// TIA Portal V15.1 export
// export: Created 2024-05-17T05:38:36.8842157Z, ExportSetting WithDefaults, DisplayName Totally Integrated Automation Portal, DisplayVersion V15.1 Update 5, DisplayName TIA Portal Openness, DisplayVersion V15.1 Update 5, DisplayName SINAMICS Startdrive Advanced, DisplayVersion V15.1, DisplayName G130, G150, S120, S150, SINAMICS MV, S210, DisplayVersion V15.1, DisplayName G110M, G120, G120C, G120D, G120P, DisplayVersion V15.1, DisplayName STEP 7 Professional, DisplayVersion V15.1 Update 5, DisplayName STEP 7 Safety, DisplayVersion V15.1, DisplayName WinCC Professional, DisplayVersion V15.1 Update 5, DisplayName SIMATIC Visualization Architect, DisplayVersion V15.1
FUNCTION_BLOCK "LGBSEW-MoviFitFCPN"   // FB6620, FBD
TITLE = LSEW-MoviFitFCPN
{ S7_Optimized_Access := 'TRUE' }
AUTHOR : ENGIE
FAMILY : Actuator
VERSION : 0.1
// ============================================================================
// This module is the interface to a SEW drive MOVIFIT FC using telegram 003
// ============================================================================
// 
// SEW drive config:
// 
//  - 8.. Unit functions
//                   l - 87 Process data assignment
// 
//                                                                    _____________________
// 870 Setpoint description PO1              l Control word 2          v l
//                                                                    _____________________
// 871 Setpoint description PO2              l Setpoint speed [%]  v l
//                                                                    _____________________
// 872 Setpoint description PO3              l Ramp                          v l
//                                                                    _____________________
// 873 Actual value description PI1         l Status word 1            v l
//                                                                    _____________________
// 874 Actual value description PI2         l Output current          v l
//                                                                    _____________________
// 875 Actual value description PI3         l Status word 2            v l
//                                                                    _____________________
// 876 PO data enable                               l Yes                               v l 
//                                                                                      l
//                                                                                      v
//                                       This changes to no when a POx paramater is changed
//                                                 Dot not forget to put this back to yes !
// stored: AutoNumber false, IsIECCheckEnabled false, IsRetainMemResEnabled false, MemoryReserve 100, SetENOAutomatically False, UDAEnableTagReadback false
   VAR_INPUT
      I_ContolInhibit { ExternalAccessible := 'False'; ExternalVisible := 'False'; ExternalWritable := 'False'} : Bool;   // Inhibit motor (disable output stage, uncontolled stop)
      I_OFF1 { ExternalAccessible := 'False'; ExternalVisible := 'False'; ExternalWritable := 'False'} : Bool;   // start / stop motor
      I_OFF2 { ExternalAccessible := 'False'; ExternalVisible := 'False'; ExternalWritable := 'False'} : Bool := True;   // OFF2 rapid stop
      I_ResetFault { ExternalAccessible := 'False'; ExternalVisible := 'False'; ExternalWritable := 'False'} : Bool;   // Reset fault
      I_BrakeRelease { ExternalAccessible := 'False'; ExternalVisible := 'False'; ExternalWritable := 'False'} : Bool;   // Command brake release
      I_ParameterSet { ExternalAccessible := 'False'; ExternalVisible := 'False'; ExternalWritable := 'False'} : Bool;   // Select parameter set
      I_SetpointSpeed { ExternalAccessible := 'False'; ExternalVisible := 'False'; ExternalWritable := 'False'} : Real;   // Setpoint speed in -100-0-100%
      I_Ramp { ExternalAccessible := 'False'; ExternalVisible := 'False'; ExternalWritable := 'False'} : Time := T#1s;   // Ramp send in miliseconds (range : 100-10000ms, if 0 then default 1s will be used)
   END_VAR
   VAR_OUTPUT
      O_DriveReady { ExternalAccessible := 'False'; ExternalVisible := 'False'; ExternalWritable := 'False'} : Bool;   // Drive ready
      O_OutputStageEnabled { ExternalAccessible := 'False'; ExternalVisible := 'False'; ExternalWritable := 'False'} : Bool;   // Inverter output stage is enabled
      O_MaintenanceSwitch { ExternalAccessible := 'False'; ExternalVisible := 'False'; ExternalWritable := 'False'} : Bool;   // Maintenance switch activated (1=mains OFF)
      O_ParameterSet { ExternalAccessible := 'False'; ExternalVisible := 'False'; ExternalWritable := 'False'} : Bool;   // Active parameter set
      O_PODataEnabled { ExternalAccessible := 'False'; ExternalVisible := 'False'; ExternalWritable := 'False'} : Bool;   // Process data is enabled (1 = Drive can be controlled via fieldbus)
      O_Fault { ExternalAccessible := 'False'; ExternalVisible := 'False'; ExternalWritable := 'False'} : Bool;   // Fault present
      O_Brake { ExternalAccessible := 'False'; ExternalVisible := 'False'; ExternalWritable := 'False'} : Bool;   // Brake status
      O_ActorVoltageOverloadDO00 { ExternalAccessible := 'False'; ExternalVisible := 'False'; ExternalWritable := 'False'} : Bool;   // Short circuit / overload of the actuator voltage for digital output DO00
      O_ActorVoltageOverloadDO01 { ExternalAccessible := 'False'; ExternalVisible := 'False'; ExternalWritable := 'False'} : Bool;   // Short circuit / overload of the actuator voltage for digital output DO01
      O_ActorVoltageOverloadDO02 { ExternalAccessible := 'False'; ExternalVisible := 'False'; ExternalWritable := 'False'} : Bool;   // Short circuit / overload of the actuator voltage for digital output DO02
      O_ActorVoltageOverloadDO03 { ExternalAccessible := 'False'; ExternalVisible := 'False'; ExternalWritable := 'False'} : Bool;   // Short circuit / overload of the actuator voltage for digital output DO03
      O_SensorVoltageOverloadGroup1 { ExternalAccessible := 'False'; ExternalVisible := 'False'; ExternalWritable := 'False'} : Bool;   // Short circuit / overload of the sensor suuply group 1 (VO24-I)
      O_SensorVoltageOverloadGroup2 { ExternalAccessible := 'False'; ExternalVisible := 'False'; ExternalWritable := 'False'} : Bool;   // Short circuit / overload of the sensor suuply group 2 (VO24-I)
      O_SensorVoltageOverloadGroup3 { ExternalAccessible := 'False'; ExternalVisible := 'False'; ExternalWritable := 'False'} : Bool;   // Short circuit / overload of the sensor suuply group 3 (VO24-I)
      O_SensorVoltageOverloadGroup4 { ExternalAccessible := 'False'; ExternalVisible := 'False'; ExternalWritable := 'False'} : Bool;   // Short circuit / overload of the sensor suuply group 4 (VO24-I)
      "O_Undervoltage24V-S" { ExternalAccessible := 'False'; ExternalVisible := 'False'; ExternalWritable := 'False'} : Bool;   // Value falls below the power limit for the actuator voltage DO00-03
      "O_InverterVoltageNotApplied24V-P" { ExternalAccessible := 'False'; ExternalVisible := 'False'; ExternalWritable := 'False'} : Bool;   // Presence of 24V_P for integrated inverter (FC) or external MOVIMOT (1=24V_P not present)
      O_MOVIFITSystemFault { ExternalAccessible := 'False'; ExternalVisible := 'False'; ExternalWritable := 'False'} : Bool;   // MOVIFIT system fault
      H_StatusWord1 { ExternalAccessible := 'False'; ExternalVisible := 'False'; ExternalWritable := 'False'} : Word;   // Status word 1 from drive
      H_StatusWord2 { ExternalAccessible := 'False'; ExternalVisible := 'False'; ExternalWritable := 'False'} : Word;   // Status word 2 from drive
      H_StatusWord3 { ExternalAccessible := 'False'; ExternalVisible := 'False'; ExternalWritable := 'False'} : Word;   // Status word 3 from drive
      H_ControlWord { ExternalAccessible := 'False'; ExternalVisible := 'False'; ExternalWritable := 'False'} : Word;   // Control word to drive
      H_SetpointSpeed { ExternalAccessible := 'False'; ExternalVisible := 'False'; ExternalWritable := 'False'} : Word;   // Speed setpoint for drive
      H_SetpointSpeedProCent { ExternalAccessible := 'False'; ExternalVisible := 'False'; ExternalWritable := 'False'} : Real;   // Speed setpoint for drive % / Speed setpoint for drive
      H_SetpointRamp { ExternalAccessible := 'False'; ExternalVisible := 'False'; ExternalWritable := 'False'} : Int;   // Ramp setpoint for drive
      H_ActualCurrentA { ExternalAccessible := 'False'; ExternalVisible := 'False'; ExternalWritable := 'False'} : Real;   // Actual current Ampere
      H_ActualCurrentProCent { ExternalAccessible := 'False'; ExternalVisible := 'False'; ExternalWritable := 'False'} : Real;   // Actual current %
      H_ActualWarning { ExternalAccessible := 'False'; ExternalVisible := 'False'; ExternalWritable := 'False'} : Int;   // Actual Warning From Drive
      H_ActualFault { ExternalAccessible := 'False'; ExternalVisible := 'False'; ExternalWritable := 'False'} : Int;   // Actual Fault From Drive
   END_VAR
   VAR_IN_OUT
      C_HWSubInput { ExternalAccessible := 'False'; ExternalVisible := 'False'; ExternalWritable := 'False'} : HW_SUBMODULE;   // Inputs telegram 3 Hardware identifier
      C_HWSubInputStatus { ExternalAccessible := 'False'; ExternalVisible := 'False'; ExternalWritable := 'False'} : HW_SUBMODULE;   // Status telegram MOVIFIT Hardware identifier
      C_HWSubOutput { ExternalAccessible := 'False'; ExternalVisible := 'False'; ExternalWritable := 'False'} : HW_SUBMODULE;   // Outputs telegram 3 Hardware identifier
      C_DriveCurrent { ExternalAccessible := 'False'; ExternalVisible := 'False'; ExternalWritable := 'False'} : Real;   // Reference current of the drive
      C_MotorCurrent { ExternalAccessible := 'False'; ExternalVisible := 'False'; ExternalWritable := 'False'} : Real;   // Reference current of the motor
   END_VAR
   VAR
      InputTelegram { ExternalAccessible := 'False'; ExternalVisible := 'False'; ExternalWritable := 'False'} : Struct   // Inputs telegram 3
         PI1 { ExternalAccessible := 'False'; ExternalVisible := 'False'; ExternalWritable := 'False'} : Struct   // Status word 1
            Status { ExternalAccessible := 'False'; ExternalVisible := 'False'; ExternalWritable := 'False'} : Byte;   // Status / error code
            OutputStageEnabled { ExternalAccessible := 'False'; ExternalVisible := 'False'; ExternalWritable := 'False'} : Bool;   // Inverter output stage is enabled
            InverterReady { ExternalAccessible := 'False'; ExternalVisible := 'False'; ExternalWritable := 'False'} : Bool;   // Inverter power section is ready for operation
            PODataEnabled { ExternalAccessible := 'False'; ExternalVisible := 'False'; ExternalWritable := 'False'} : Bool;   // Process data is enabled (1 = Drive can be controlled via fieldbus)
            Spare1 { ExternalAccessible := 'False'; ExternalVisible := 'False'; ExternalWritable := 'False'} : Bool;   // Reserved / not used
            CurrentParSet { ExternalAccessible := 'False'; ExternalVisible := 'False'; ExternalWritable := 'False'} : Bool;   // Current parameter set
            FaultWarning { ExternalAccessible := 'False'; ExternalVisible := 'False'; ExternalWritable := 'False'} : Bool;   // Fault/warning present
            Spare2 { ExternalAccessible := 'False'; ExternalVisible := 'False'; ExternalWritable := 'False'} : Bool;   // Reserved / not used
            Spare3 { ExternalAccessible := 'False'; ExternalVisible := 'False'; ExternalWritable := 'False'} : Bool;   // Reserved / not used
         END_STRUCT;
         Current { ExternalAccessible := 'False'; ExternalVisible := 'False'; ExternalWritable := 'False'} : Int;   // Current
         PI3 { ExternalAccessible := 'False'; ExternalVisible := 'False'; ExternalWritable := 'False'} : Struct   // Status word 2
            brake { ExternalAccessible := 'False'; ExternalVisible := 'False'; ExternalWritable := 'False'} : Bool;   // Brake released
            Spare4 { ExternalAccessible := 'False'; ExternalVisible := 'False'; ExternalWritable := 'False'} : Bool;   // Reserved / not used
            Spare5 { ExternalAccessible := 'False'; ExternalVisible := 'False'; ExternalWritable := 'False'} : Bool;   // Reserved / not used
            Spare6 { ExternalAccessible := 'False'; ExternalVisible := 'False'; ExternalWritable := 'False'} : Bool;   // Reserved / not used
            Spare7 { ExternalAccessible := 'False'; ExternalVisible := 'False'; ExternalWritable := 'False'} : Bool;   // Reserved / not used
            Spare8 { ExternalAccessible := 'False'; ExternalVisible := 'False'; ExternalWritable := 'False'} : Bool;   // Reserved / not used
            Spare9 { ExternalAccessible := 'False'; ExternalVisible := 'False'; ExternalWritable := 'False'} : Bool;   // Reserved / not used
            Spare10 { ExternalAccessible := 'False'; ExternalVisible := 'False'; ExternalWritable := 'False'} : Bool;   // Reserved / not used
            OutputStageEnabled { ExternalAccessible := 'False'; ExternalVisible := 'False'; ExternalWritable := 'False'} : Bool;   // Inverter output stage is enabled
            InverterReady { ExternalAccessible := 'False'; ExternalVisible := 'False'; ExternalWritable := 'False'} : Bool;   // Inverter power section is ready for operation
            PODataEnabled { ExternalAccessible := 'False'; ExternalVisible := 'False'; ExternalWritable := 'False'} : Bool;   // Process data is enabled (1 = Drive can be controlled via fieldbus)
            Spare11 { ExternalAccessible := 'False'; ExternalVisible := 'False'; ExternalWritable := 'False'} : Bool;   // Reserved / not used
            CurrentParSet { ExternalAccessible := 'False'; ExternalVisible := 'False'; ExternalWritable := 'False'} : Bool;   // Current parameter set
            FaultWarning { ExternalAccessible := 'False'; ExternalVisible := 'False'; ExternalWritable := 'False'} : Bool;   // Fault/warning present
            Spare12 { ExternalAccessible := 'False'; ExternalVisible := 'False'; ExternalWritable := 'False'} : Bool;   // Reserved / not used
            Spare13 { ExternalAccessible := 'False'; ExternalVisible := 'False'; ExternalWritable := 'False'} : Bool;   // Reserved / not used
         END_STRUCT;
      END_STRUCT;
      InputStatusTelegram { ExternalAccessible := 'False'; ExternalVisible := 'False'; ExternalWritable := 'False'} : Struct   // Status telegram MOVIFIT
         ActorVoltageOverloadDO00 { ExternalAccessible := 'False'; ExternalVisible := 'False'; ExternalWritable := 'False'} : Bool;   // Short circuit / overload of the actuator voltage for digital output DO00
         ActorVoltageOverloadDO01 { ExternalAccessible := 'False'; ExternalVisible := 'False'; ExternalWritable := 'False'} : Bool;   // Short circuit / overload of the actuator voltage for digital output DO01
         ActorVoltageOverloadDO02 { ExternalAccessible := 'False'; ExternalVisible := 'False'; ExternalWritable := 'False'} : Bool;   // Short circuit / overload of the actuator voltage for digital output DO02
         ActorVoltageOverloadDO03 { ExternalAccessible := 'False'; ExternalVisible := 'False'; ExternalWritable := 'False'} : Bool;   // Short circuit / overload of the actuator voltage for digital output DO03
         SensorVoltageOverloadGroup1 { ExternalAccessible := 'False'; ExternalVisible := 'False'; ExternalWritable := 'False'} : Bool;   // Short circuit / overload of the sensor suuply group 1 (VO24-I)
         SensorVoltageOverloadGroup2 { ExternalAccessible := 'False'; ExternalVisible := 'False'; ExternalWritable := 'False'} : Bool;   // Short circuit / overload of the sensor suuply group 2 (VO24-I)
         SensorVoltageOverloadGroup3 { ExternalAccessible := 'False'; ExternalVisible := 'False'; ExternalWritable := 'False'} : Bool;   // Short circuit / overload of the sensor suuply group 3 (VO24-I)
         SensorVoltageOverloadGroup4 { ExternalAccessible := 'False'; ExternalVisible := 'False'; ExternalWritable := 'False'} : Bool;   // Short circuit / overload of the sensor suuply group 4 (VO24-I)
         MaintenanceSwitch { ExternalAccessible := 'False'; ExternalVisible := 'False'; ExternalWritable := 'False'} : Bool;   // Maintenance switch activated (1=mains OFF)
         "Undervoltage24V-S" { ExternalAccessible := 'False'; ExternalVisible := 'False'; ExternalWritable := 'False'} : Bool;   // Value falls below the power limit for the actuator voltage DO00-03
         "InverterVoltageNotApplied24V-P" { ExternalAccessible := 'False'; ExternalVisible := 'False'; ExternalWritable := 'False'} : Bool;   // Presence of 24V_P for integrated inverter (FC) or external MOVIMOT (1=24V_P not present)
         Spare1 { ExternalAccessible := 'False'; ExternalVisible := 'False'; ExternalWritable := 'False'} : Bool;   // Reserved / not used
         Spare2 { ExternalAccessible := 'False'; ExternalVisible := 'False'; ExternalWritable := 'False'} : Bool;   // Reserved / not used
         Spare3 { ExternalAccessible := 'False'; ExternalVisible := 'False'; ExternalWritable := 'False'} : Bool;   // Reserved / not used
         Spare4 { ExternalAccessible := 'False'; ExternalVisible := 'False'; ExternalWritable := 'False'} : Bool;   // Reserved / not used
         MOVIFITSystemFault { ExternalAccessible := 'False'; ExternalVisible := 'False'; ExternalWritable := 'False'} : Bool;   // MOVIFIT system fault
      END_STRUCT;
      OutputTelegram { ExternalAccessible := 'False'; ExternalVisible := 'False'; ExternalWritable := 'False'} : Struct   // Outputs telegram 3
         PO1 { ExternalAccessible := 'False'; ExternalVisible := 'False'; ExternalWritable := 'False'} : Struct
            BrakeRelease { ExternalAccessible := 'False'; ExternalVisible := 'False'; ExternalWritable := 'False'} : Bool;   // Release brake
            CTW_Bit9 { ExternalAccessible := 'False'; ExternalVisible := 'False'; ExternalWritable := 'False'} : Bool;   // Reserved / not used
            CTW_Bit10 { ExternalAccessible := 'False'; ExternalVisible := 'False'; ExternalWritable := 'False'} : Bool;   // Reserved / not used
            CTW_Bit11 { ExternalAccessible := 'False'; ExternalVisible := 'False'; ExternalWritable := 'False'} : Bool;   // Reserved / not used
            CTW_Bit12 { ExternalAccessible := 'False'; ExternalVisible := 'False'; ExternalWritable := 'False'} : Bool;   // Reserved / not used
            CTW_Bit13 { ExternalAccessible := 'False'; ExternalVisible := 'False'; ExternalWritable := 'False'} : Bool;   // Reserved / not used
            CTW_Bit14 { ExternalAccessible := 'False'; ExternalVisible := 'False'; ExternalWritable := 'False'} : Bool;   // Reserved / not used
            CTW_Bit15 { ExternalAccessible := 'False'; ExternalVisible := 'False'; ExternalWritable := 'False'} : Bool;   // Reserved / not used
            ContrInhibit { ExternalAccessible := 'False'; ExternalVisible := 'False'; ExternalWritable := 'False'} : Bool;   // Interlock to drive
            RapidStop { ExternalAccessible := 'False'; ExternalVisible := 'False'; ExternalWritable := 'False'} : Bool;   // Rapid stop with stop ramp t13/t23, brake applied after stop
            Stop { ExternalAccessible := 'False'; ExternalVisible := 'False'; ExternalWritable := 'False'} : Bool;   // Stop to drive at normal ramp
            CTW_Bit3 { ExternalAccessible := 'False'; ExternalVisible := 'False'; ExternalWritable := 'False'} : Bool;   // Reserved / not used
            CTW_Bit4 { ExternalAccessible := 'False'; ExternalVisible := 'False'; ExternalWritable := 'False'} : Bool;   // Reserved / not used
            CTW_Bit5 { ExternalAccessible := 'False'; ExternalVisible := 'False'; ExternalWritable := 'False'} : Bool;   // Reserved / not used / Parameter set 1 or 2
            ResetFault { ExternalAccessible := 'False'; ExternalVisible := 'False'; ExternalWritable := 'False'} : Bool;   // Reset fault on drive
            CTW_Bit7 { ExternalAccessible := 'False'; ExternalVisible := 'False'; ExternalWritable := 'False'} : Bool;   // Reserved / not used
         END_STRUCT;
         SetpointSpeed { ExternalAccessible := 'False'; ExternalVisible := 'False'; ExternalWritable := 'False'} : Word;   // Speed setpoint for drive (-4000-0-4000hex)
         Ramp { ExternalAccessible := 'False'; ExternalVisible := 'False'; ExternalWritable := 'False'} : Int;   // Ramp setpoint for drive
      END_STRUCT;
   END_VAR
   VAR_TEMP
      TempReal : Real;   // Temp Real
   END_VAR
   VAR_TEMP   // added for the SCL form of the ladder/FBD networks
      _w1 : Bool;
   END_VAR
BEGIN

REGION Network 1: **** 1 - Inputs **** Read input telegram and store in struct
   // Copies the Input telegram to a local varibale struct
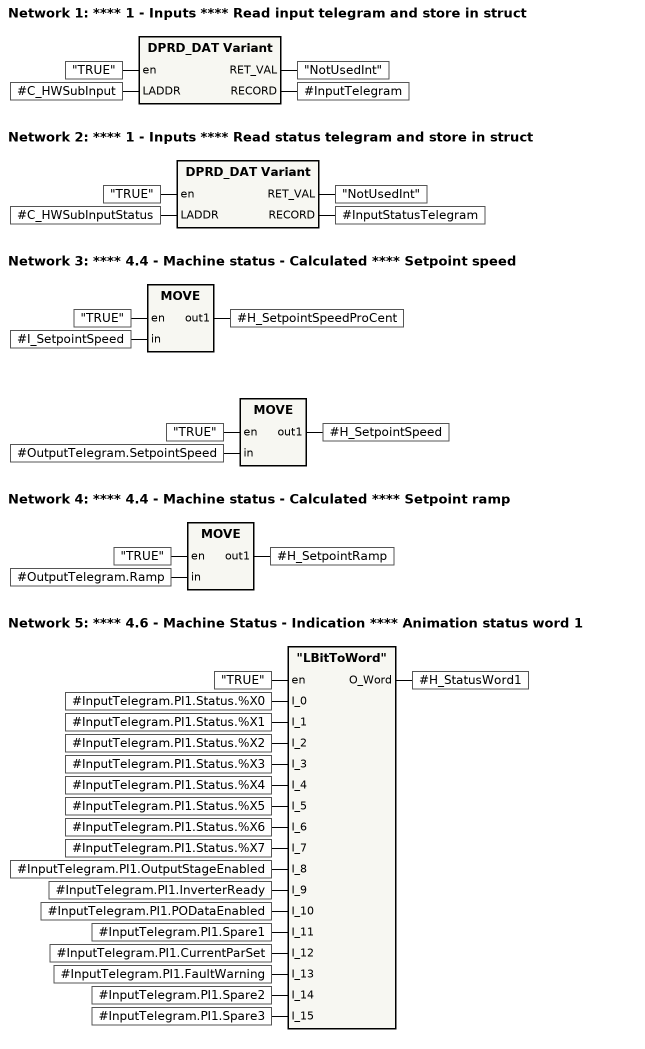
   IF "TRUE" THEN
       "NotUsedInt" := DPRD_DAT(LADDR := #C_HWSubInput, RECORD => #InputTelegram);   // Copy data with HW ID _________ /________ / l input telegram l SEW l l ===============>> PLC l Drive _l / -l__l
   END_IF;
END_REGION

REGION Network 2: **** 1 - Inputs **** Read status telegram and store in struct
   // Copies the status telegram to a local varibale struct
   IF "TRUE" THEN
       "NotUsedInt" := DPRD_DAT(LADDR := #C_HWSubInputStatus, RECORD => #InputStatusTelegram);   // Copy data with HW ID _________ /________ / l Status telegram l SEW l l ===============>> PLC l Drive _l / -l__l
   END_IF;
END_REGION

REGION Network 3: **** 4.4 - Machine status - Calculated **** Setpoint speed
   // Convert Data
   IF "TRUE" THEN
       #H_SetpointSpeedProCent := #I_SetpointSpeed;
       #H_SetpointSpeed := #OutputTelegram.SetpointSpeed;
   END_IF;
END_REGION

REGION Network 4: **** 4.4 - Machine status - Calculated **** Setpoint ramp
   // Convert Data
   IF "TRUE" THEN #H_SetpointRamp := #OutputTelegram.Ramp; END_IF;
END_REGION

REGION Network 5: **** 4.6 - Machine Status - Indication **** Animation status word 1
   // Animation
   IF "TRUE" THEN
       "LBitToWord"(I_0 := #InputTelegram.PI1.Status.%X0,
                    I_1 := #InputTelegram.PI1.Status.%X1,
                    I_2 := #InputTelegram.PI1.Status.%X2,
                    I_3 := #InputTelegram.PI1.Status.%X3,
                    I_4 := #InputTelegram.PI1.Status.%X4,
                    I_5 := #InputTelegram.PI1.Status.%X5,
                    I_6 := #InputTelegram.PI1.Status.%X6,
                    I_7 := #InputTelegram.PI1.Status.%X7,
                    I_8 := #InputTelegram.PI1.OutputStageEnabled,
                    I_9 := #InputTelegram.PI1.InverterReady,
                    I_10 := #InputTelegram.PI1.PODataEnabled,
                    I_11 := #InputTelegram.PI1.Spare1,
                    I_12 := #InputTelegram.PI1.CurrentParSet,
                    I_13 := #InputTelegram.PI1.FaultWarning,
                    I_14 := #InputTelegram.PI1.Spare2,
                    I_15 := #InputTelegram.PI1.Spare3,
                    O_Word => #H_StatusWord1);
   END_IF;
END_REGION

REGION Network 6: **** 4.6 - Machine Status - Indication **** Animation status word 2
   // Animation
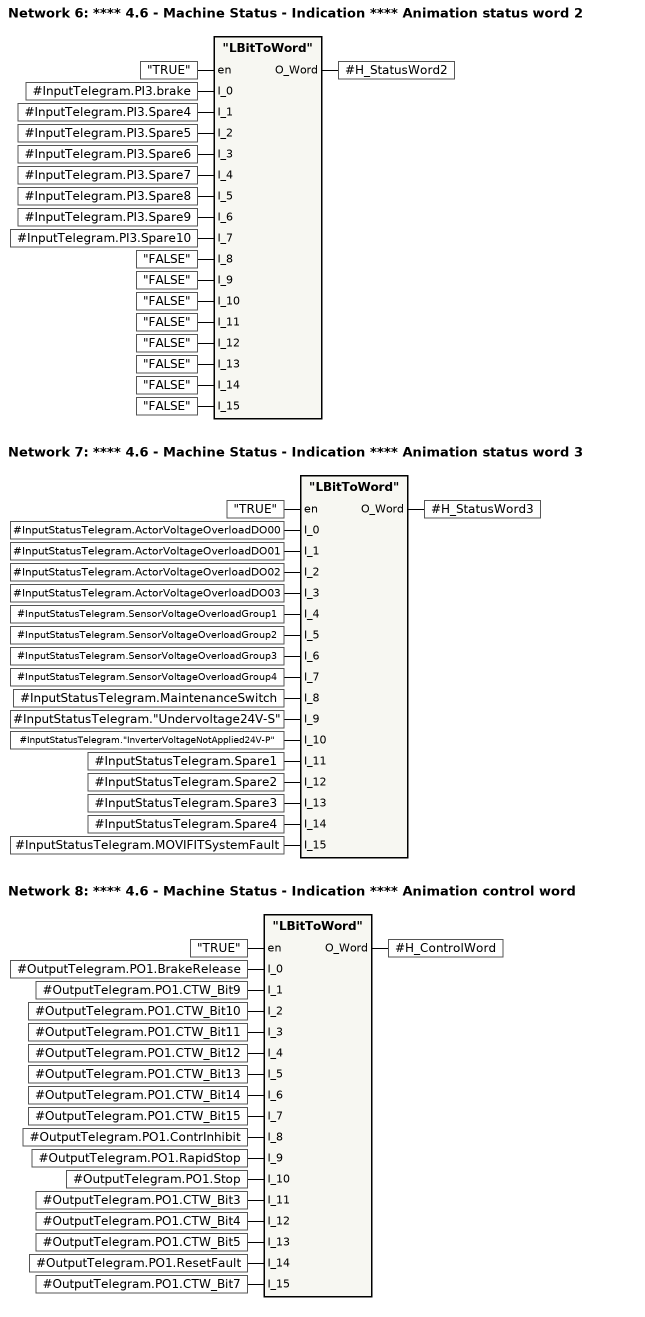
   IF "TRUE" THEN
       "LBitToWord"(I_0 := #InputTelegram.PI3.brake,
                    I_1 := #InputTelegram.PI3.Spare4,
                    I_2 := #InputTelegram.PI3.Spare5,
                    I_3 := #InputTelegram.PI3.Spare6,
                    I_4 := #InputTelegram.PI3.Spare7,
                    I_5 := #InputTelegram.PI3.Spare8,
                    I_6 := #InputTelegram.PI3.Spare9,
                    I_7 := #InputTelegram.PI3.Spare10,
                    I_8 := "FALSE",
                    I_9 := "FALSE",
                    I_10 := "FALSE",
                    I_11 := "FALSE",
                    I_12 := "FALSE",
                    I_13 := "FALSE",
                    I_14 := "FALSE",
                    I_15 := "FALSE",
                    O_Word => #H_StatusWord2);
   END_IF;
END_REGION

REGION Network 7: **** 4.6 - Machine Status - Indication **** Animation status word 3
   // Animation
   IF "TRUE" THEN
       "LBitToWord"(I_0 := #InputStatusTelegram.ActorVoltageOverloadDO00,
                    I_1 := #InputStatusTelegram.ActorVoltageOverloadDO01,
                    I_2 := #InputStatusTelegram.ActorVoltageOverloadDO02,
                    I_3 := #InputStatusTelegram.ActorVoltageOverloadDO03,
                    I_4 := #InputStatusTelegram.SensorVoltageOverloadGroup1,
                    I_5 := #InputStatusTelegram.SensorVoltageOverloadGroup2,
                    I_6 := #InputStatusTelegram.SensorVoltageOverloadGroup3,
                    I_7 := #InputStatusTelegram.SensorVoltageOverloadGroup4,
                    I_8 := #InputStatusTelegram.MaintenanceSwitch,
                    I_9 := #InputStatusTelegram."Undervoltage24V-S",
                    I_10 := #InputStatusTelegram."InverterVoltageNotApplied24V-P",
                    I_11 := #InputStatusTelegram.Spare1,
                    I_12 := #InputStatusTelegram.Spare2,
                    I_13 := #InputStatusTelegram.Spare3,
                    I_14 := #InputStatusTelegram.Spare4,
                    I_15 := #InputStatusTelegram.MOVIFITSystemFault,
                    O_Word => #H_StatusWord3);
   END_IF;
END_REGION

REGION Network 8: **** 4.6 - Machine Status - Indication **** Animation control word
   // Animation
   IF "TRUE" THEN
       "LBitToWord"(I_0 := #OutputTelegram.PO1.BrakeRelease,
                    I_1 := #OutputTelegram.PO1.CTW_Bit9,
                    I_2 := #OutputTelegram.PO1.CTW_Bit10,
                    I_3 := #OutputTelegram.PO1.CTW_Bit11,
                    I_4 := #OutputTelegram.PO1.CTW_Bit12,
                    I_5 := #OutputTelegram.PO1.CTW_Bit13,
                    I_6 := #OutputTelegram.PO1.CTW_Bit14,
                    I_7 := #OutputTelegram.PO1.CTW_Bit15,
                    I_8 := #OutputTelegram.PO1.ContrInhibit,
                    I_9 := #OutputTelegram.PO1.RapidStop,
                    I_10 := #OutputTelegram.PO1.Stop,
                    I_11 := #OutputTelegram.PO1.CTW_Bit3,
                    I_12 := #OutputTelegram.PO1.CTW_Bit4,
                    I_13 := #OutputTelegram.PO1.CTW_Bit5,
                    I_14 := #OutputTelegram.PO1.ResetFault,
                    I_15 := #OutputTelegram.PO1.CTW_Bit7,
                    O_Word => #H_ControlWord);
   END_IF;
END_REGION

REGION Network 9: **** 4.6 - Machine Status - Calculated **** Status / Warning / Fault code from drive
   // When the fault input is "True"   then the status code send over the byte is a fault code as decimal.
   // When the fault input is "False" then the status code send over the byte is a warning / status code as decimal.
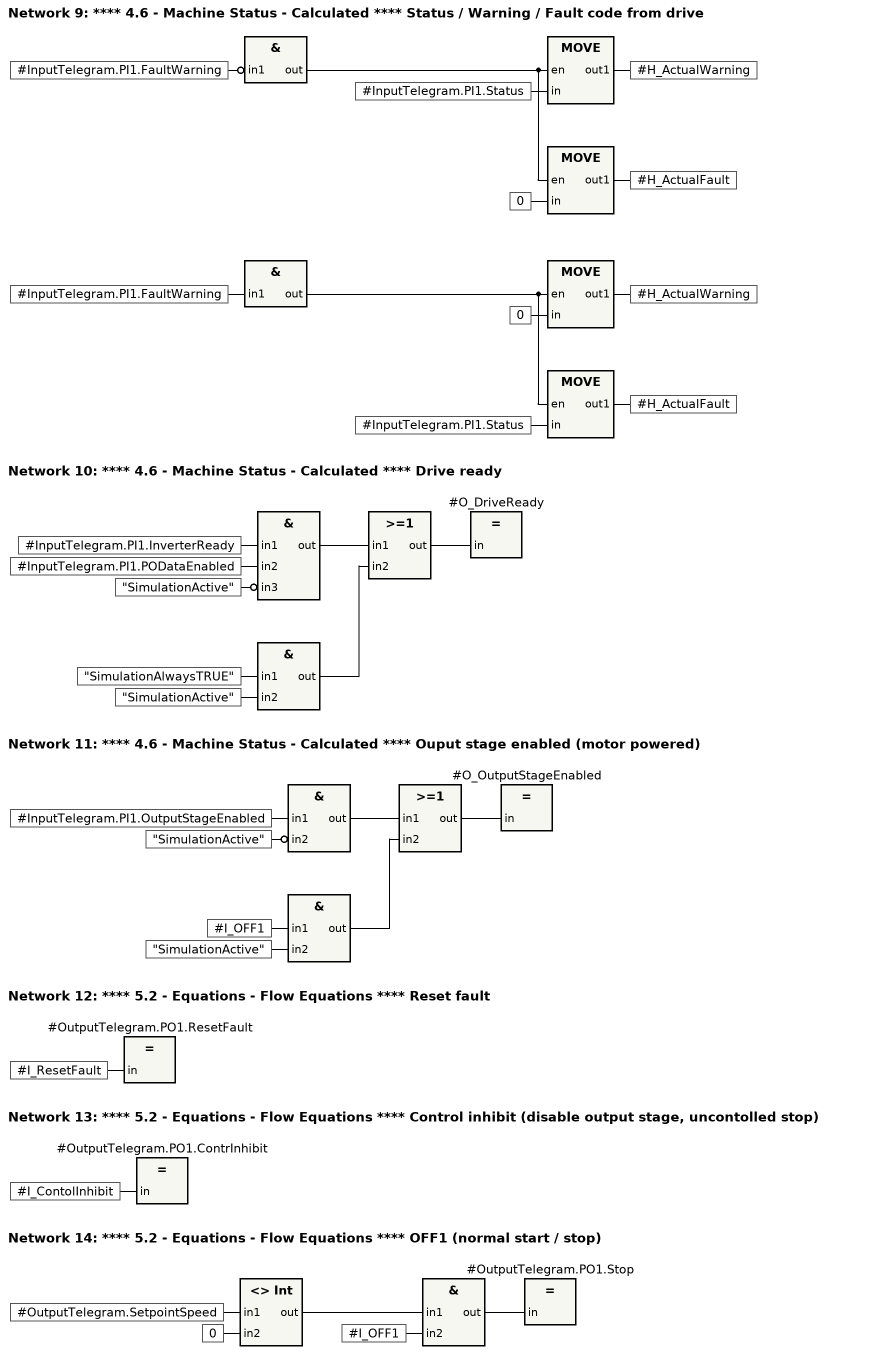
   IF NOT #InputTelegram.PI1.FaultWarning THEN
       #H_ActualWarning := #InputTelegram.PI1.Status;
       #H_ActualFault := 0;
   END_IF;
   IF #InputTelegram.PI1.FaultWarning THEN
       #H_ActualWarning := 0;
       #H_ActualFault := #InputTelegram.PI1.Status;
   END_IF;
END_REGION

REGION Network 10: **** 4.6 - Machine Status - Calculated **** Drive ready
   // Drive ready state and process data from PLC is active (Drive is listening to PLC)
   #O_DriveReady := (#InputTelegram.PI1.InverterReady AND #InputTelegram.PI1.PODataEnabled AND NOT "SimulationActive") OR ("SimulationAlwaysTRUE" AND "SimulationActive");
END_REGION

REGION Network 11: **** 4.6 - Machine Status - Calculated **** Ouput stage enabled (motor powered)
   // Ouput stage enabled (motor powered)
   #O_OutputStageEnabled := (#InputTelegram.PI1.OutputStageEnabled AND NOT "SimulationActive") OR (#I_OFF1 AND "SimulationActive");
END_REGION

REGION Network 12: **** 5.2 - Equations - Flow Equations **** Reset fault
   #OutputTelegram.PO1.ResetFault := #I_ResetFault;
END_REGION

REGION Network 13: **** 5.2 - Equations - Flow Equations **** Control inhibit (disable output stage, uncontolled stop)
   #OutputTelegram.PO1.ContrInhibit := #I_ContolInhibit;
END_REGION

REGION Network 14: **** 5.2 - Equations - Flow Equations **** OFF1 (normal start / stop)
   #OutputTelegram.PO1.Stop := (#OutputTelegram.SetpointSpeed <> 0) AND #I_OFF1;
END_REGION

REGION Network 15: **** 5.2 - Equations - Flow Equations **** OFF2 (rapid stop)
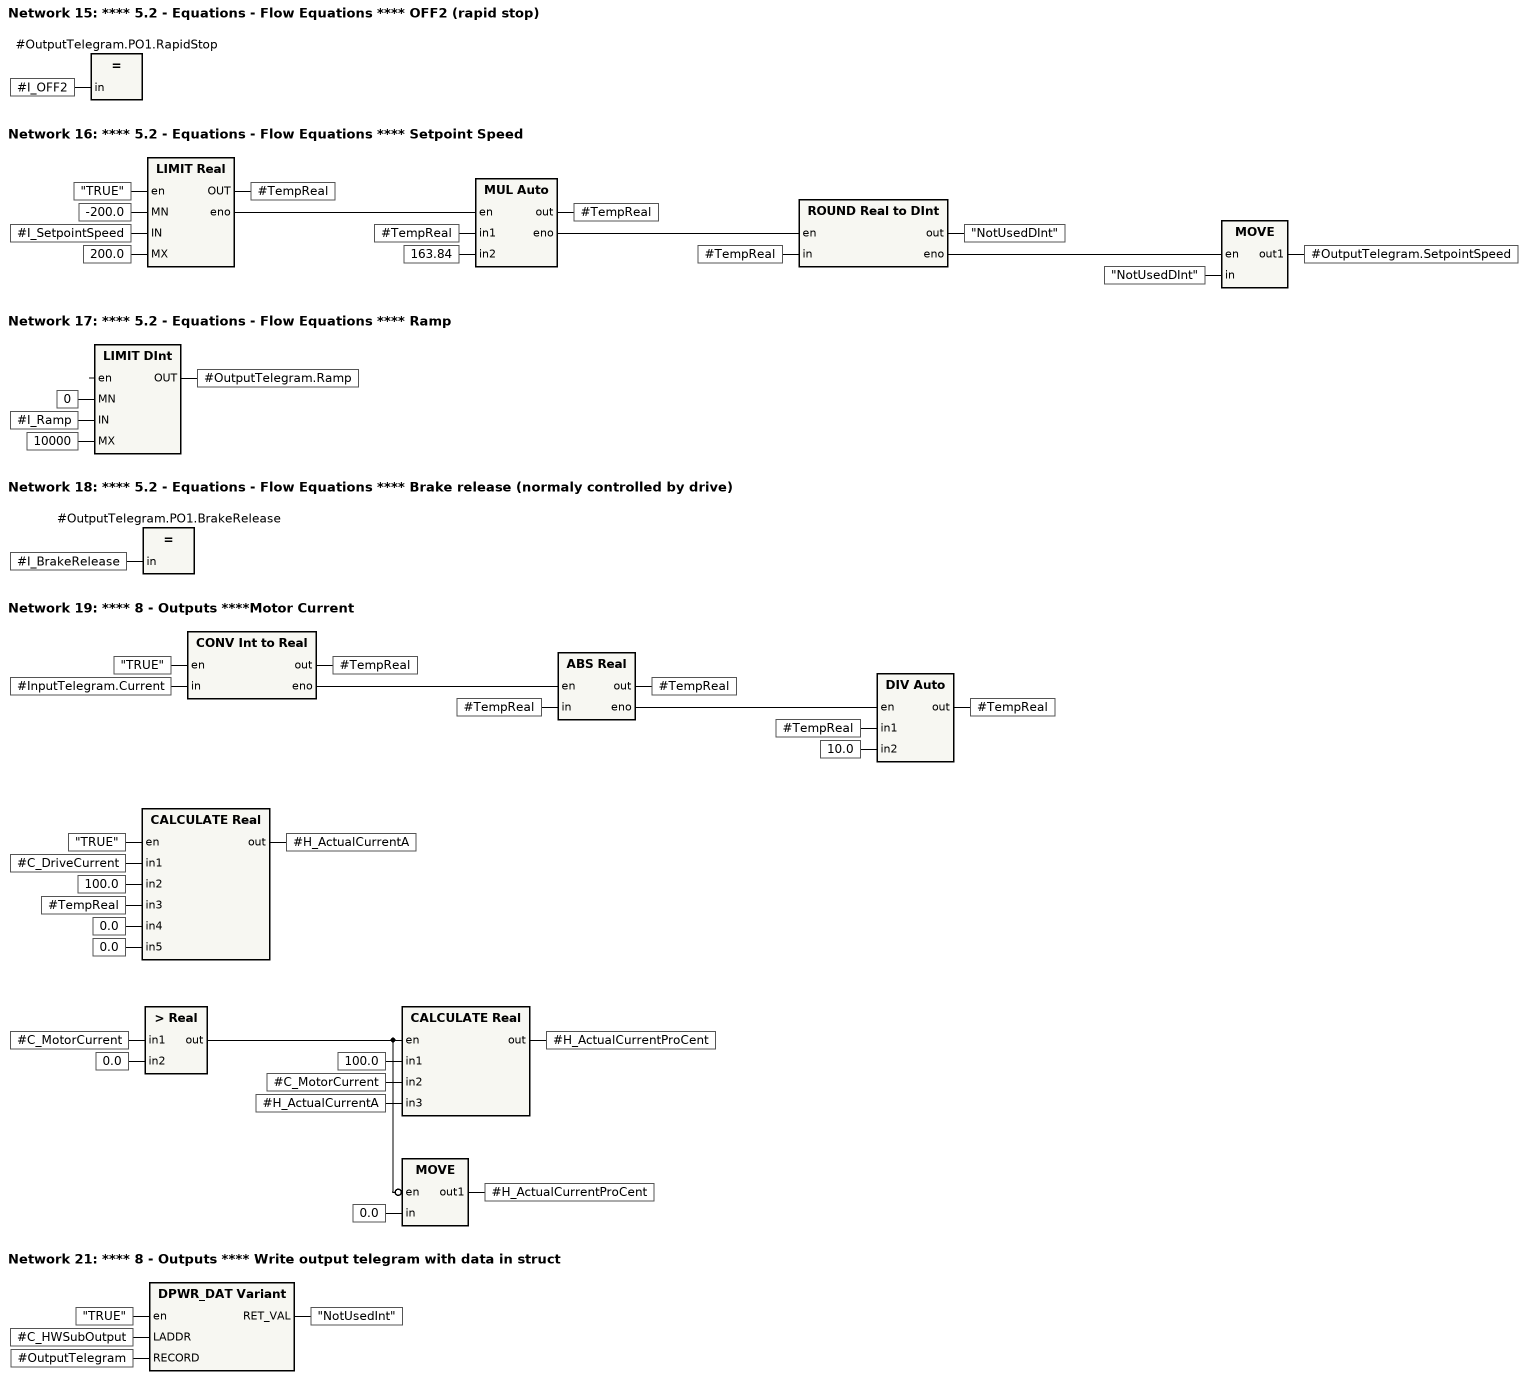
   #OutputTelegram.PO1.RapidStop := #I_OFF2;   // ^ Speed (%) Stop signal at 5s l / 100% l______________/_ l \ \ l \ \ l \ \ l \ \ 0% l___________________\_____\___________________________> Time (s) l OFF2 OFF1 (regular start stop) 7s 10s Ramp down time settings to be done in the drive. OFF2 is to be used for controlled stops when there is a need to stop faster then regular, for example when there is an E-stop at a lift it is better to do a conttrolled stop and after that (x time in safety program) to give a STO. Note if there is a safe stop availible on safety level this is to be used instead of the non safety signals. _
END_REGION

REGION Network 16: **** 5.2 - Equations - Flow Equations **** Setpoint Speed
   // Setpoint to drive is given in 0 to 4000Hex = 0 to 100% of maximum speed / 
   //                                                   0 to -4000Hex  = 0 to -100% of maximum speed.
   // 
   // maximum speed is not the same as motor reference speed!
   // 
   // 4000Hex = 16384 dec.
   IF "TRUE" THEN
       #TempReal := LIMIT(MN := -200.0, IN := #I_SetpointSpeed, MX := 200.0);   // Limit input setpiont from -200 to 200%
       #TempReal := #TempReal * 163.84;   // Convert: -100-0-100% to -4000-0-4000Hex -16384-0-16384 dec. _
       "NotUsedDInt" := ROUND(#TempReal);
       #OutputTelegram.SetpointSpeed := "NotUsedDInt";
   END_IF;
END_REGION

REGION Network 17: **** 5.2 - Equations - Flow Equations **** Ramp
   // Ramp send in miliseconds (range : 100-10000ms, if 0 then default 1s will be used)
   #OutputTelegram.Ramp := LIMIT(MN := 0, IN := #I_Ramp, MX := 10000);   // Speed The ramp up / down time is (Rpm) ^ / set with this parameter l _________ / l / \/ l / \ l____/ \____ l--------------------------------------------------> t (s) _
END_REGION

REGION Network 18: **** 5.2 - Equations - Flow Equations **** Brake release (normaly controlled by drive)
   // Brake release (normaly controlled by drive), Possibility to release brake at any moment.
   #OutputTelegram.PO1.BrakeRelease := #I_BrakeRelease;   // Not to be used for normal operation!!! In normal operation this is done by the drive.
END_REGION

REGION Network 19: **** 8 - Outputs ****Motor Current
   // Motor Current in % compared to the drive reference current (not the motor reference current)
   IF "TRUE" THEN
       #TempReal := INT_TO_REAL(#InputTelegram.Current);
       #TempReal := ABS(#TempReal);   // Motor Current in % compared to the drive reference current (not the motor reference current) Remove - sign and use absolute value. Then scale this to the correct value (divide by 10 to get %) (This needs to be done since the drive can only send intiger values and not real values, so the drive does the percentage x10 to give a value behind the comma.) Then scale the % to a Ampere value and a % value compared to the motor reference current.
       #TempReal := #TempReal / 10.0;
       #H_ActualCurrentA := #C_DriveCurrent - (((100.0 - #TempReal) / (100.0 - 0.0)) * (#C_DriveCurrent- 0.0));
   END_IF;
   #_w1 := #C_MotorCurrent > 0.0;
   IF #_w1 THEN #H_ActualCurrentProCent := (100.0 / #C_MotorCurrent) * #H_ActualCurrentA; END_IF;
   IF NOT #_w1 THEN #H_ActualCurrentProCent := 0.0; END_IF;
END_REGION

REGION Network 20 (SCL): **** 8 - Outputs **** Status / Fault booleans
   // Copy input telegram booleans to O_****** parameters for use outside this block.

   #O_ParameterSet := #InputTelegram.PI1.CurrentParSet;
   #O_PODataEnabled := #InputTelegram.PI1.PODataEnabled;
   #O_Fault := #InputTelegram.PI1.FaultWarning;
   IF NOT "SimulationActive" THEN
       #O_Brake := #InputTelegram.PI3.brake;
   ELSE
       #O_Brake := "SimulationAlwaysTRUE";
   END_IF;
   #O_MaintenanceSwitch := #InputStatusTelegram.MaintenanceSwitch;
   #O_ActorVoltageOverloadDO00 := #InputStatusTelegram.ActorVoltageOverloadDO00;
   #O_ActorVoltageOverloadDO01 := #InputStatusTelegram.ActorVoltageOverloadDO01;
   #O_ActorVoltageOverloadDO02 := #InputStatusTelegram.ActorVoltageOverloadDO02;
   #O_ActorVoltageOverloadDO03 := #InputStatusTelegram.ActorVoltageOverloadDO03;
   #O_SensorVoltageOverloadGroup1 := #InputStatusTelegram.SensorVoltageOverloadGroup1;
   #O_SensorVoltageOverloadGroup2 := #InputStatusTelegram.SensorVoltageOverloadGroup2;
   #O_SensorVoltageOverloadGroup3 := #InputStatusTelegram.SensorVoltageOverloadGroup3;
   #O_SensorVoltageOverloadGroup4 := #InputStatusTelegram.SensorVoltageOverloadGroup4;
   #"O_Undervoltage24V-S" := #InputStatusTelegram."Undervoltage24V-S";
   #"O_InverterVoltageNotApplied24V-P" := #InputStatusTelegram."InverterVoltageNotApplied24V-P";
   #O_MOVIFITSystemFault := #InputStatusTelegram.MOVIFITSystemFault;
END_REGION

REGION Network 21: **** 8 - Outputs **** Write output telegram with data in struct
   IF "TRUE" THEN
       "NotUsedInt" := DPWR_DAT(LADDR := #C_HWSubOutput, RECORD := #OutputTelegram);   // Copy data with HW ID _________ output telegram /________ / l PLC ===============>> l SEW l l l Drive _l / -l__l
   END_IF;
END_REGION
END_FUNCTION_BLOCK
